// Frequence to time(PT is Timer target value)
FUNCTION F_FtoPT : Time
VAR_INPUT
	Hz : REAL;
END_VAR
VAR
END_VAR

IF Hz > 0 THEN
	F_FtoPT := DWORD_TO_TIME(REAL_TO_DWORD((1000 / Hz)));
ELSE
	F_FtoPT := T#0S;
END_IF

END_FUNCTION

(* stored: Version 1.1.0.1, ProductVersion 3.1.4024.13
   POU F_FtoPT: Id {fdc4ca46-1de8-4a96-89a4-03039d84ba57}, SpecialFunc None *)
